{attribute addProperty BoxType "EL2595-0000-0018"}
{attribute addProperty Id "OutputBIT10.1252Input_trigger_enableBIT10.1254ResetBIT10.1258"}
{attribute addProperty CRC "1704927272"}
{attribute addProperty SizeInBites "16"}
{attribute addProperty SizeInBytes "2"}
TYPE Control_659F2028 :
STRUCT
	{attribute 'hide'}
	reserve_1 : BIT;
	{attribute addProperty Name "Output"}
	Output : BIT;
	{attribute 'hide'}
	reserve_2 : BIT;
	{attribute addProperty Name "Input_trigger_enable"}
	Input_trigger_enable : BIT;
	{attribute 'hide'}
	reserve_3_BIT_0 : BIT;
	{attribute 'hide'}
	reserve_3_BIT_1 : BIT;
	{attribute 'hide'}
	reserve_3_BIT_2 : BIT;
	{attribute addProperty Name "Reset"}
	Reset : BIT;
	{attribute 'hide'}
	reserve_4 : BYTE;
END_STRUCT
END_TYPE

(* stored: Version 1.2.0.0, ProductVersion 3.1.4024.9
   DUT Control_659F2028: Id {16d1d9ef-2d52-4fbe-806f-fdcb21ffa265} *)
